FUNCTION F_LminToEng : LREAL
VAR_INPUT
	fLmin : LREAL;
END_VAR
VAR
END_VAR

F_LminToEng := fLmin / 60000;

END_FUNCTION

(* stored: Version 1.1.0.1, ProductVersion 3.1.4024.10
   POU F_LminToEng: Id {cbf5fe98-cab1-4eb5-ae30-ba273c87a7ec}, SpecialFunc None *)
